(* CODESYS project Simulator.ecp

Project tree, tasks and I/O mapping:
  Controller : 750-8214 PFC200 G2 2ETH RS CAN, WAGO, order no. 0750-8214, version 5.17.3.10
    application Application
      libraries: 
      task PLC_Task (cyclic, interval t#50ms, priority 15) calls Simulator
      task VISU_TASK (cyclic, interval 100 ms, priority 15) calls VisuElems.Visu_Prg
      program Simulator [LD]
      Functionblocks/
        function block Arduino [ST]
        function block UR10 [ST]
        function block Wago1 [ST]
        function block Wago2 [ST]
      global variables Sim
      visualisation Simulator
    Kbus : Kbus, WAGO, version 1.4.0.2
        unmapped channels: K-BUS diagnostics
    MODBUS
      MODBUS : MODBUS, WAGO, order no. n/a, version 1.1.1.16
    CANbus
    Common.PCI
    EtherNet/IP
      Ethernet : Ethernet, WAGO, version 35.17.0.0
    Serial
      COM1 : COM1, WAGO, version 0.0.0.19
  libraries: VisuSymbols, 4.1.0.0 (System); WagoVisuIcons, 1.1.0.5 (WAGO)
  text list GlobalTextList
*)

// Controller/Application/Sim
{attribute 'qualified_only'}
VAR_GLOBAL
	Encoder : INT;
	Robot_Degrees : INT;
	Robot_Degrees_UR10_Base : INT;
	Robot_Degrees_UR10_Sholder : INT;
	Robot_Degrees_UR10_Elbow : INT;
	Robot_Degrees_UR10_Wrist1 : INT;
	Robot_Degrees_UR10_Wrist2 : INT;
	Robot_Degrees_UR10_Wrist3 : INT;
	
	Encoder_Base : INT;
	Encoder_Sholder : INT;
	Encoder_Elbow : INT;
	Encoder_Wrist1 : INT;
	Encoder_Wrist2 : INT;
	Encoder_Wrist3 : INT;
	
	Base : INT;
	Sholder : INT;
	Elbow : INT;
	Wrist1 : INT;
	Wrist2 : INT;
	Wrist3 : INT;
	
	
END_VAR

// Controller/Application/Simulator
PROGRAM Simulator
VAR
	Arduino_0: Arduino;
	Wago1_0: Wago1;
	UR10_0: UR10;
	Wago2_0: Wago2;
END_VAR

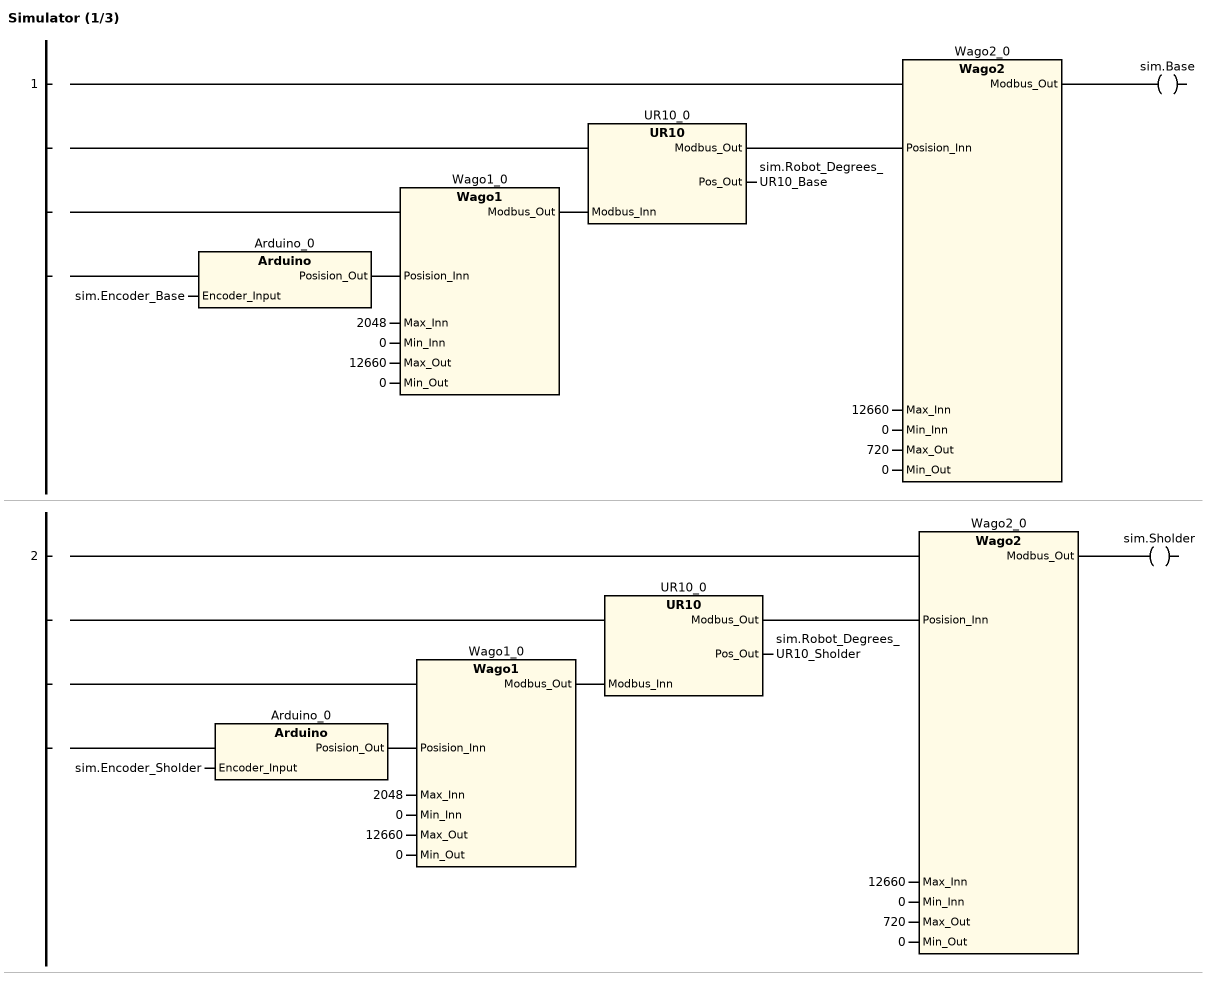
// NETWORK 1
Arduino_0(Encoder_Input := sim.Encoder_Base); // Arduino
Wago1_0(
    Posision_Inn := Arduino_0.Posision_Out,
    Max_Inn := 2048,
    Min_Inn := 0,
    Max_Out := 12660,
    Min_Out := 0); // Wago1
UR10_0(Modbus_Inn := Wago1_0.Modbus_Out, Pos_Out => sim.Robot_Degrees_UR10_Base); // UR10
Wago2_0(Posision_Inn := UR10_0.Modbus_Out, Max_Inn := 12660, Min_Inn := 0, Max_Out := 720, Min_Out := 0); // Wago2
sim.Base := Wago2_0.Modbus_Out;

// NETWORK 2
Arduino_0(Encoder_Input := sim.Encoder_Sholder); // Arduino
Wago1_0(
    Posision_Inn := Arduino_0.Posision_Out,
    Max_Inn := 2048,
    Min_Inn := 0,
    Max_Out := 12660,
    Min_Out := 0); // Wago1
UR10_0(Modbus_Inn := Wago1_0.Modbus_Out, Pos_Out => sim.Robot_Degrees_UR10_Sholder); // UR10
Wago2_0(Posision_Inn := UR10_0.Modbus_Out, Max_Inn := 12660, Min_Inn := 0, Max_Out := 720, Min_Out := 0); // Wago2
sim.Sholder := Wago2_0.Modbus_Out;

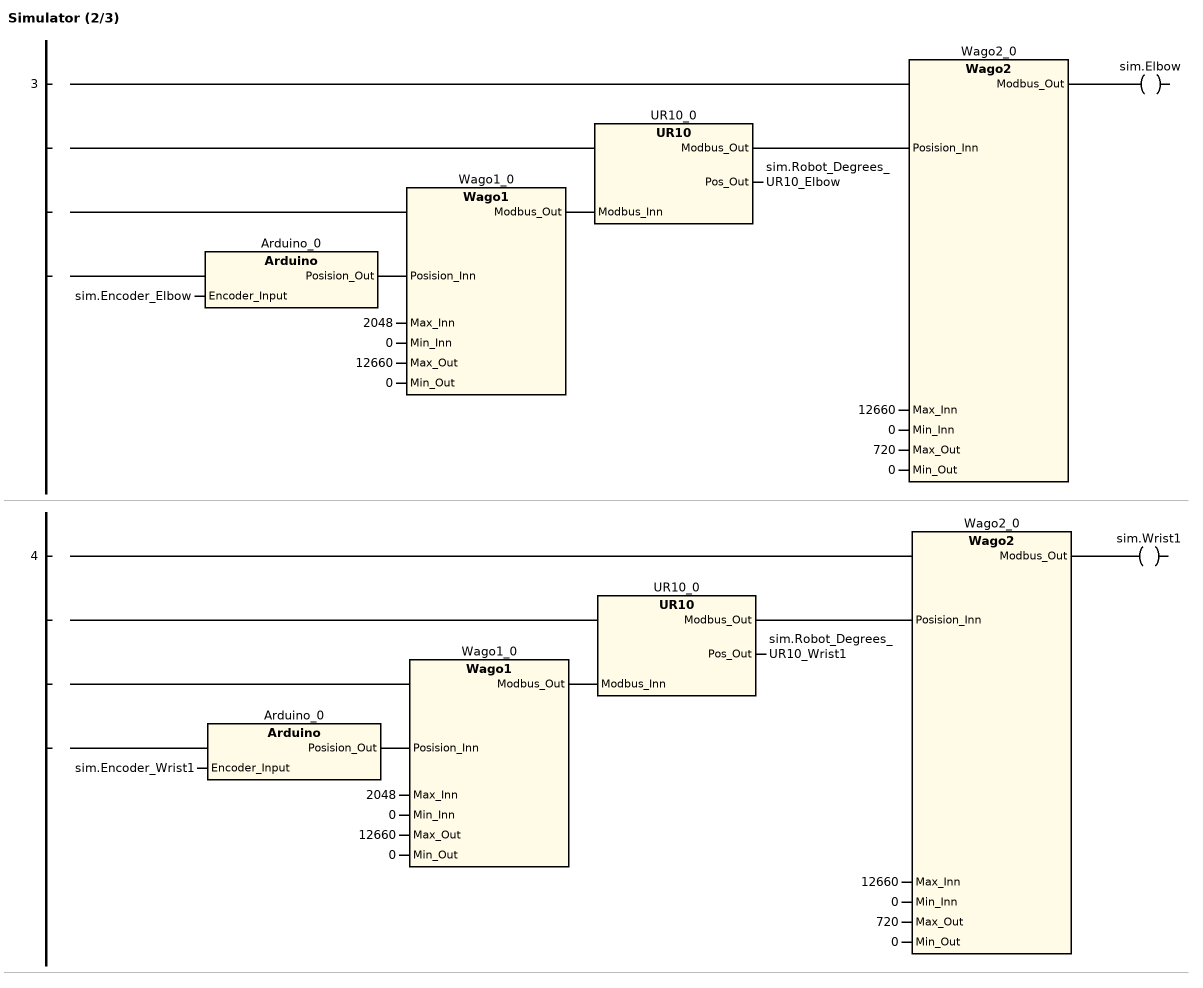
// NETWORK 3
Arduino_0(Encoder_Input := sim.Encoder_Elbow); // Arduino
Wago1_0(
    Posision_Inn := Arduino_0.Posision_Out,
    Max_Inn := 2048,
    Min_Inn := 0,
    Max_Out := 12660,
    Min_Out := 0); // Wago1
UR10_0(Modbus_Inn := Wago1_0.Modbus_Out, Pos_Out => sim.Robot_Degrees_UR10_Elbow); // UR10
Wago2_0(Posision_Inn := UR10_0.Modbus_Out, Max_Inn := 12660, Min_Inn := 0, Max_Out := 720, Min_Out := 0); // Wago2
sim.Elbow := Wago2_0.Modbus_Out;

// NETWORK 4
Arduino_0(Encoder_Input := sim.Encoder_Wrist1); // Arduino
Wago1_0(
    Posision_Inn := Arduino_0.Posision_Out,
    Max_Inn := 2048,
    Min_Inn := 0,
    Max_Out := 12660,
    Min_Out := 0); // Wago1
UR10_0(Modbus_Inn := Wago1_0.Modbus_Out, Pos_Out => sim.Robot_Degrees_UR10_Wrist1); // UR10
Wago2_0(Posision_Inn := UR10_0.Modbus_Out, Max_Inn := 12660, Min_Inn := 0, Max_Out := 720, Min_Out := 0); // Wago2
sim.Wrist1 := Wago2_0.Modbus_Out;

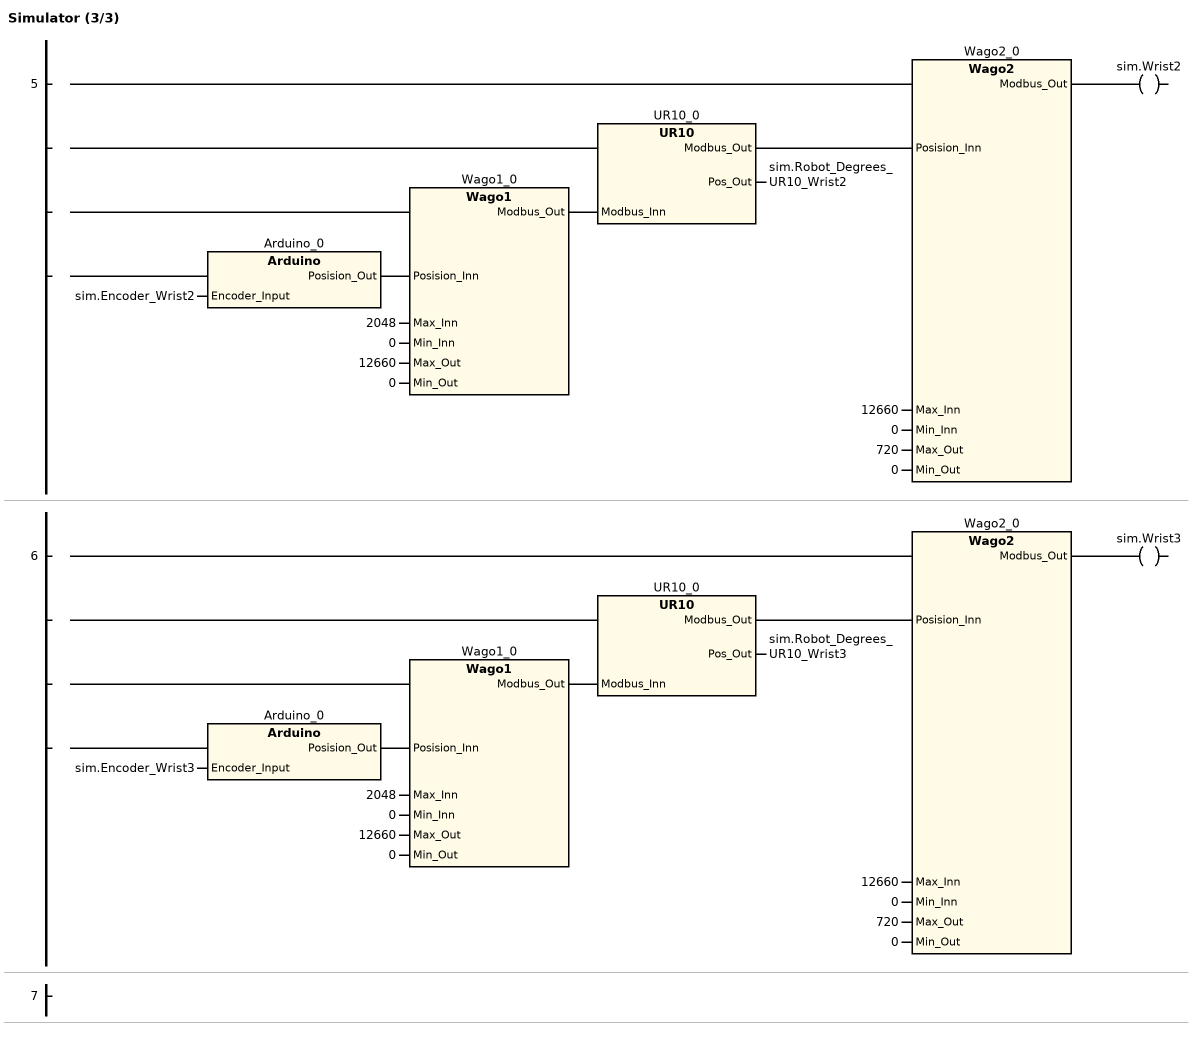
// NETWORK 5
Arduino_0(Encoder_Input := sim.Encoder_Wrist2); // Arduino
Wago1_0(
    Posision_Inn := Arduino_0.Posision_Out,
    Max_Inn := 2048,
    Min_Inn := 0,
    Max_Out := 12660,
    Min_Out := 0); // Wago1
UR10_0(Modbus_Inn := Wago1_0.Modbus_Out, Pos_Out => sim.Robot_Degrees_UR10_Wrist2); // UR10
Wago2_0(Posision_Inn := UR10_0.Modbus_Out, Max_Inn := 12660, Min_Inn := 0, Max_Out := 720, Min_Out := 0); // Wago2
sim.Wrist2 := Wago2_0.Modbus_Out;

// NETWORK 6
Arduino_0(Encoder_Input := sim.Encoder_Wrist3); // Arduino
Wago1_0(
    Posision_Inn := Arduino_0.Posision_Out,
    Max_Inn := 2048,
    Min_Inn := 0,
    Max_Out := 12660,
    Min_Out := 0); // Wago1
UR10_0(Modbus_Inn := Wago1_0.Modbus_Out, Pos_Out => sim.Robot_Degrees_UR10_Wrist3); // UR10
Wago2_0(Posision_Inn := UR10_0.Modbus_Out, Max_Inn := 12660, Min_Inn := 0, Max_Out := 720, Min_Out := 0); // Wago2
sim.Wrist3 := Wago2_0.Modbus_Out;

// NETWORK 7

END_PROGRAM

// Controller/Application/Functionblocks/Wago2
FUNCTION_BLOCK Wago2
VAR_INPUT
	Posision_Inn : INT;
	Max_Inn : REAL;
	Min_Inn : REAL;
	Max_Out : REAL;
	Min_Out : REAL;
END_VAR
VAR_OUTPUT
	Modbus_Out : INT;
END_VAR
VAR
	Posision : REAL;
	RadPos : REAL;
END_VAR

Posision := INT_TO_REAL(Posision_Inn);

RadPos := Posision * ((Max_Out - Min_Out)/(Max_Inn - Min_Inn));

Modbus_Out := REAL_TO_INT(RadPos-360);

END_FUNCTION_BLOCK

// Controller/Application/Functionblocks/UR10
FUNCTION_BLOCK UR10
VAR_INPUT
	Modbus_Inn : INT;
END_VAR
VAR_OUTPUT
	Modbus_Out : INT;
	Pos_Out : INT;
END_VAR
VAR
	Rad : REAL;
	Rad2 : REAL;
	Degree : REAL;
	Mod_In : REAL;
	Mod_Out : REAL;
END_VAR

Mod_In := INT_TO_REAL(Modbus_inn);

Rad := ((Mod_In/1000)-6.28);
Degree := (Rad * (180/3.1415));

IF Rad < -6.28
	THEN Rad := -6.28;
END_IF

IF Rad > 6.28
	THEN Rad := 6.28;
END_IF

Pos_Out := REAL_TO_INT(Degree);

Rad2 := ((Rad+6.28)*1000);

Modbus_Out := Real_To_INT(Rad2);

END_FUNCTION_BLOCK

// Controller/Application/Functionblocks/Wago1
FUNCTION_BLOCK Wago1
VAR_INPUT
	Posision_Inn : INT;
	Max_Inn : REAL;
	Min_Inn : REAL;
	Max_Out : REAL;
	Min_Out : REAL;
END_VAR
VAR_OUTPUT
	Modbus_Out : INT;
END_VAR
VAR
	Posision : REAL;
	RadPos : REAL;
END_VAR

Posision := INT_TO_REAL(Posision_Inn);

RadPos := Posision * ((Max_Out - Min_Out)/(Max_Inn - Min_Inn));

Modbus_Out := REAL_TO_INT(RadPos);

END_FUNCTION_BLOCK

// Controller/Application/Functionblocks/Arduino
FUNCTION_BLOCK Arduino
VAR_INPUT
	Encoder_Input : INT;
END_VAR
VAR_OUTPUT
	Posision_Out : INT;
END_VAR
VAR
END_VAR

Posision_Out := Encoder_Input;

END_FUNCTION_BLOCK

// Controller/Application/Simulator
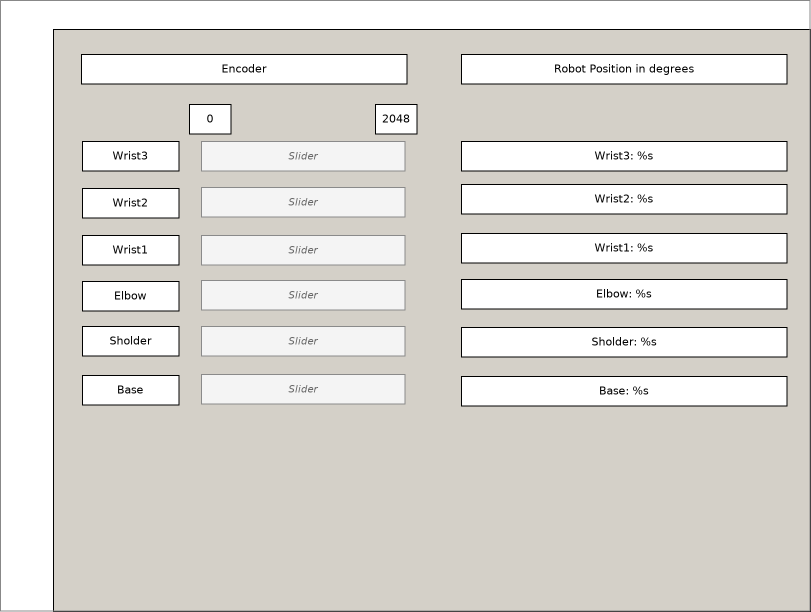
VISUALIZATION Simulator  // 811x612
    Rectangle (53,29 758x583)
    Rectangle (81,54 326x30), "Encoder"
    Rectangle (461,54 326x30), "Robot Position in degrees"
    Slider (201,141 204x30), variable: Sim.Encoder_Wrist3, scale 0..2048
    Slider (201,187 204x30), variable: Sim.Encoder_Wrist2, scale 0..2048
    Slider (201,235 204x30), variable: Sim.Encoder_Wrist1, scale 0..2048
    Slider (201,280 204x30), variable: Sim.Encoder_Elbow, scale 0..2048
    Slider (201,326 204x30), variable: Sim.Encoder_Sholder, scale 0..2048
    Slider (201,374 204x30), variable: Sim.Encoder_Base, scale 0..2048
    Rectangle (82,141 97x30), "Wrist3"
    Rectangle (82,188 97x30), "Wrist2"
    Rectangle (82,235 97x30), "Wrist1"
    Rectangle (82,281 97x30), "Elbow"
    Rectangle (82,326 97x30), "Sholder"
    Rectangle (82,375 97x30), "Base"
    Rectangle (189,104 42x30), "0"
    Rectangle (375,104 42x30), "2048"
    Rectangle (461,141 326x30), "Wrist3: %s", text variable: Sim.Wrist3
    Rectangle (461,184 326x30), "Wrist2: %s", text variable: Sim.Wrist2
    Rectangle (461,233 326x30), "Wrist1: %s", text variable: Sim.Wrist1
    Rectangle (461,279 326x30), "Elbow: %s", text variable: Sim.Elbow
    Rectangle (461,327 326x30), "Sholder: %s", text variable: Sim.Sholder
    Rectangle (461,376 326x30), "Base: %s", text variable: Sim.Base
END_VISUALIZATION
